// TIA Portal project "2022.06.10_温度模块" (V17)

(* hardware
DEVICE "S7-1200 station_1"  S7-1200 Station
   slot 0: "Rack_0"  S7-1200 Rack  Rack  V1.0
   slot 1: "PLC_1"  CPU 1212C DC/DC/DC  6ES7 212-1AE40-0XB0  V4.5
   slot 2: "AI 4xRTD_1"  SM 1231 AI4 x RTD  6ES7 231-5PD32-0XB0  V2.0
*)

// ===== PLC "PLC_1"  CPU 1212C DC/DC/DC =====

VAR_GLOBAL   // PLC tag table "默认变量表"
   "Tag_1" AT %IW96 : Word;
   "Tag_2" AT %MD40 : DWord;
   "Tag_3" AT %MD44 : UDInt;
END_VAR

ORGANIZATION_BLOCK "Main"   // OB1, LAD, ProgramCycle
TITLE = "Main Program Sweep (Cycle)"
{ S7_Optimized_Access := 'TRUE' }
VERSION : 0.1
   VAR_INPUT
      Initial_Call : Bool;   // Initial call of this OB
      Remanence : Bool;   // =True, if remanent data are available
   END_VAR
BEGIN

REGION Network 1
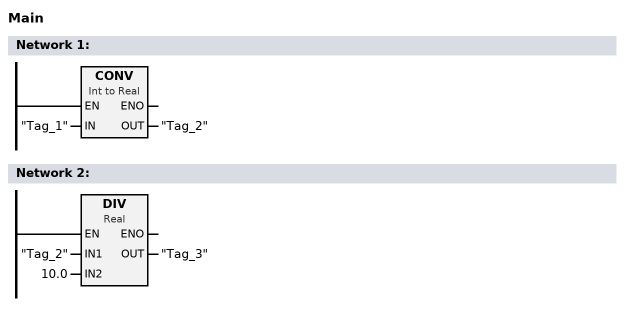
   RUNG wire#powerrail
      { S7_Templates := "[SrcType := Int, DestType := Real]" } Convert(in := "Tag_1", out => "Tag_2")
   END_RUNG
   // the same network as SCL:
   "Tag_2" := INT_TO_REAL("Tag_1");
END_REGION

REGION Network 2
   RUNG wire#powerrail
      { S7_Templates := "SrcType := Real" } Div(in1 := "Tag_2", in2 := 10.0, out => "Tag_3")
   END_RUNG
   // the same network as SCL:
   "Tag_3" := "Tag_2" / 10.0;
END_REGION
END_ORGANIZATION_BLOCK